{attribute 'GeneratedUsingTerminal: KL3182'}
{attribute addProperty BoxType "KL3182"}
{attribute addProperty Description ""}
{attribute addProperty Physics ""}
{attribute addProperty Id "Channel_1AT %Q*Channel_6576A6810Channel_2AT %Q*Channel_6576A6810"}
{attribute addProperty CRC "2957383796"}
{attribute addProperty Size "0"}
TYPE KL3182_B0461874 :
STRUCT
	{attribute addProperty Name "Channel_1"}
	Channel_1 : Channel_6576A681;
	{attribute addProperty Name "Channel_2"}
	Channel_2 : Channel_6576A681;
END_STRUCT
END_TYPE

(* stored: Version 1.2.0.0, ProductVersion 3.1.4024.9
   DUT KL3182_B0461874: Id {2ba844c4-6822-4d54-8cdd-b38d606a2085} *)
